FUNCTION MF_Singleton : real
VAR_INPUT
	x,a:REAL;
END_VAR
VAR
END_VAR

IF x=a then
	MF_Singleton:=1;
ELSE
	MF_Singleton:=0;
END_IF

END_FUNCTION

(* stored: Version 1.1.0.1, ProductVersion 3.1.4024.6
   POU MF_Singleton: Id {46a49336-bd84-4f42-9f86-16245c3b9aaa}, SpecialFunc None *)
